FUNCTION_BLOCK IMREAD (* Imread OpenCV function block *)
  (* Version 1.0, AN, SWDC RTSoft *)
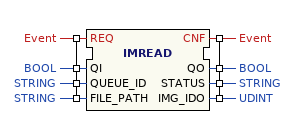
  EVENT_INPUT
    REQ WITH QI, QUEUE_ID, FILE_PATH;
  END_EVENT
  EVENT_OUTPUT
    CNF WITH QO, STATUS, IMG_IDO;
  END_EVENT
  VAR_INPUT
    QI : BOOL;
    QUEUE_ID : STRING;
    FILE_PATH : STRING;
  END_VAR
  VAR_OUTPUT
    QO : BOOL;
    STATUS : STRING;
    IMG_IDO : UDINT;
  END_VAR
  (* Service APPLICATION/RESOURCE: Service Interface Function Block Type *)
END_FUNCTION_BLOCK
